// TIA Portal V20 export
DATA_BLOCK "气缸面板多路复用变量"   // DB11
{ S7_Optimized_Access := 'TRUE' }
// stored: MemoryReserve 100
   VAR
      Valve_index : "VALVE_HMI_UDT";
      HMI_Positon_X24 { S7_SetPoint := 'True'} : Bool;
   END_VAR
BEGIN
END_DATA_BLOCK
